GLOBALCONSTANTS myPorts (* Global constants *)
  (* Standard: 61499-1 *)
  (* Version 1.0, 2023-10-22, franz *)
  VAR_GLOBAL CONSTANT
    PORT_0 : WSTRING := "fbdk[].ip[239.0.0.1:61000]";
    PORT_1 : WSTRING := "fbdk[].ip[239.0.0.1:61001]";
    PORT_2 : WSTRING := "fbdk[].ip[239.0.0.1:61002]";
    PORT_3 : WSTRING := "fbdk[].ip[239.0.0.1:61003]";
    PORT_A0 : WSTRING := "fbdk[].ip[localhost:61500]";
    PORT_A1 : WSTRING := "fbdk[].ip[localhost:61501]";
    PORT_A2 : WSTRING := "fbdk[].ip[localhost:61502]";
    PORT_A3 : WSTRING := "fbdk[].ip[localhost:61503]";
    PORT_B0 : WSTRING := "fbdk[].ip[192.168.178.58:61500]";
    PORT_B1 : WSTRING := "fbdk[].ip[192.168.178.58:61501]";
    PORT_B2 : WSTRING := "fbdk[].ip[192.168.178.58:61502]";
    PORT_B3 : WSTRING := "fbdk[].ip[192.168.178.58:61503]";
  END_VAR
END_GLOBALCONSTANTS
